// TIA Portal V21 export
FUNCTION "ampoule" : Void   // FC6, LAD
{ S7_Optimized_Access := 'TRUE' }
// stored: SetENOAutomatically false
   VAR_TEMP   // added for the SCL form of the ladder/FBD networks
      _w1 : Bool;
      _w2 : Bool;
   END_VAR
BEGIN

REGION Network 1
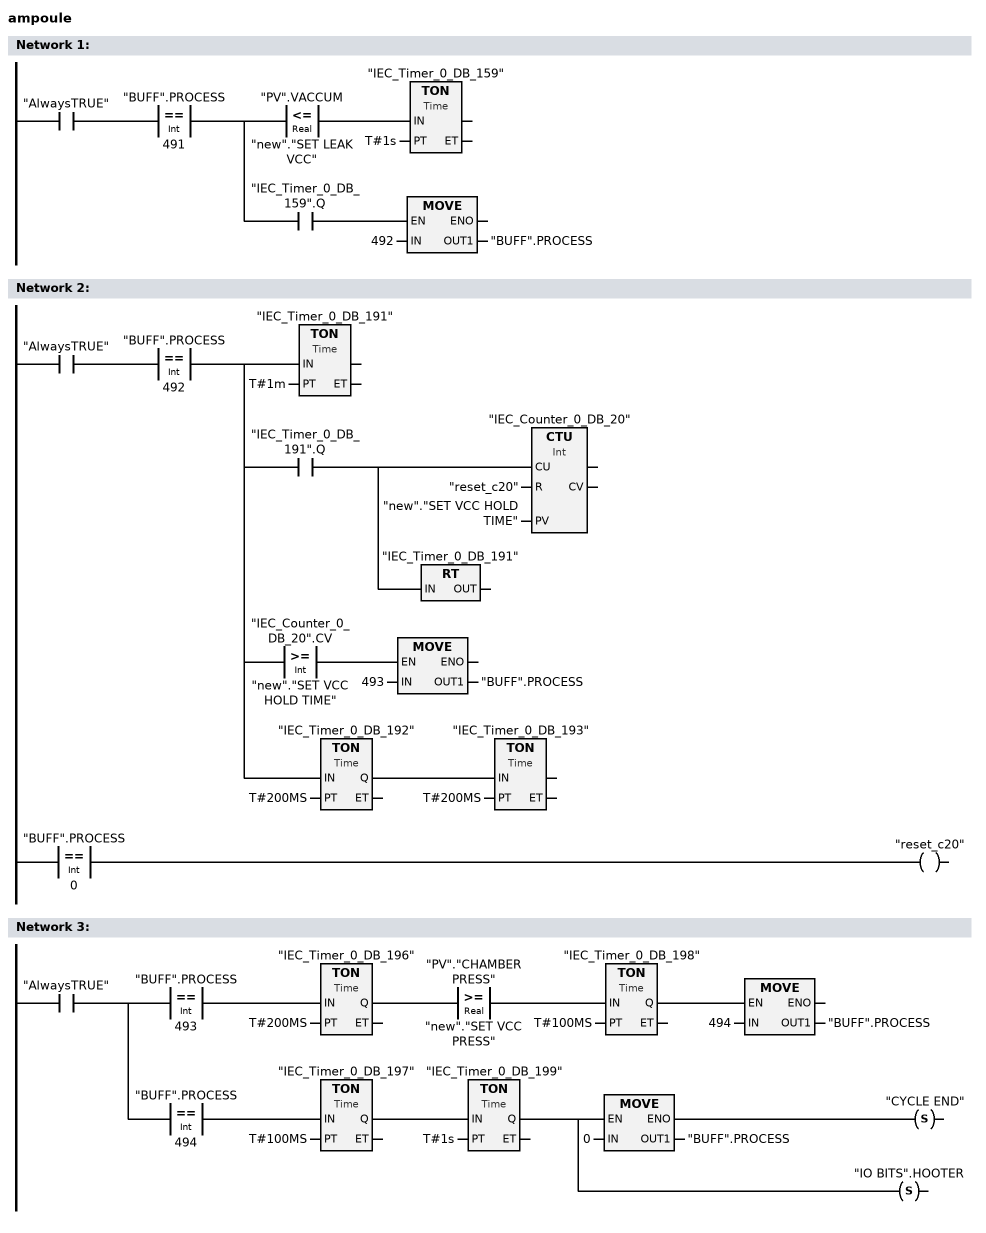
   RUNG wire#powerrail
      Contact( "AlwaysTRUE" )
      { S7_Templates := "SrcType := Int" } EQ_Contact(in1 := "BUFF".PROCESS, in2 := 491)
      wire#w1
      { S7_Templates := "SrcType := Real" } LE_Contact(in1 := "PV".VACCUM, in2 := "new"."SET LEAK VCC")
      { S7_Templates := "time_type := Time" } "IEC_Timer_0_DB_159".TON(pt := T#1s, et =>)
   END_RUNG
   RUNG wire#w1
      Contact( "IEC_Timer_0_DB_159".Q )
      Move(in := 492, out1 => "BUFF".PROCESS)
   END_RUNG
   // the same network as SCL:
   #_w1 := "AlwaysTRUE" AND ("BUFF".PROCESS = 491);
   "IEC_Timer_0_DB_159".TON(IN := #_w1 AND ("PV".VACCUM <= "new"."SET LEAK VCC"), PT := T#1s);
   IF #_w1 AND "IEC_Timer_0_DB_159".Q THEN "BUFF".PROCESS := 492; END_IF;
END_REGION

REGION Network 2
   RUNG wire#powerrail
      Contact( "AlwaysTRUE" )
      { S7_Templates := "SrcType := Int" } EQ_Contact(in1 := "BUFF".PROCESS, in2 := 492)
      wire#w1
      { S7_Templates := "time_type := Time" } "IEC_Timer_0_DB_191".TON(pt := T#1m, et =>)
   END_RUNG
   RUNG wire#w1
      Contact( "IEC_Timer_0_DB_191".Q )
      wire#w2
      { S7_Templates := "value_type := Int" } "IEC_Counter_0_DB_20".CTU(r := "reset_c20", pv := "new"."SET VCC HOLD TIME", cv =>)
   END_RUNG
   RUNG wire#w2
      RT_Coil( "IEC_Timer_0_DB_191" )
   END_RUNG
   RUNG wire#w1
      { S7_Templates := "SrcType := Int" } GE_Contact(in1 := "IEC_Counter_0_DB_20".CV, in2 := "new"."SET VCC HOLD TIME")
      Move(in := 493, out1 => "BUFF".PROCESS)
   END_RUNG
   RUNG wire#w1
      { S7_Templates := "time_type := Time" } "IEC_Timer_0_DB_192".TON(pt := T#200MS, et =>)
      { S7_Templates := "time_type := Time" } "IEC_Timer_0_DB_193".TON(pt := T#200MS, et =>)
   END_RUNG
   RUNG wire#powerrail
      { S7_Templates := "SrcType := Int" } EQ_Contact(in1 := "BUFF".PROCESS, in2 := 0)
      Coil( "reset_c20" )
   END_RUNG
   // the same network as SCL:
   #_w1 := "AlwaysTRUE" AND ("BUFF".PROCESS = 492);
   "IEC_Timer_0_DB_191".TON(IN := #_w1, PT := T#1m);
   #_w2 := #_w1 AND "IEC_Timer_0_DB_191".Q;
   "IEC_Counter_0_DB_20".CTU(CU := #_w2, R := "reset_c20", PV := "new"."SET VCC HOLD TIME");
   IF #_w2 THEN RESET_TIMER("IEC_Timer_0_DB_191"); END_IF;
   IF #_w1 AND ("IEC_Counter_0_DB_20".CV >= "new"."SET VCC HOLD TIME") THEN "BUFF".PROCESS := 493; END_IF;
   "IEC_Timer_0_DB_192".TON(IN := #_w1, PT := T#200MS);
   "IEC_Timer_0_DB_193".TON(IN := "IEC_Timer_0_DB_192".Q, PT := T#200MS);
   "reset_c20" := "BUFF".PROCESS = 0;
END_REGION

REGION Network 3
   RUNG wire#powerrail
      Contact( "AlwaysTRUE" )
      wire#w1
      { S7_Templates := "SrcType := Int" } EQ_Contact(in1 := "BUFF".PROCESS, in2 := 493)
      { S7_Templates := "time_type := Time" } "IEC_Timer_0_DB_196".TON(pt := T#200MS, et =>)
      { S7_Templates := "SrcType := Real" } GE_Contact(in1 := "PV"."CHAMBER PRESS", in2 := "new"."SET VCC PRESS")
      { S7_Templates := "time_type := Time" } "IEC_Timer_0_DB_198".TON(pt := T#100MS, et =>)
      Move(in := 494, out1 => "BUFF".PROCESS)
   END_RUNG
   RUNG wire#w1
      { S7_Templates := "SrcType := Int" } EQ_Contact(in1 := "BUFF".PROCESS, in2 := 494)
      { S7_Templates := "time_type := Time" } "IEC_Timer_0_DB_197".TON(pt := T#100MS, et =>)
      { S7_Templates := "time_type := Time" } "IEC_Timer_0_DB_199".TON(pt := T#1s, et =>)
      wire#w2
      Move(in := 0, out1 => "BUFF".PROCESS)
      S_Coil( "CYCLE END" )
   END_RUNG
   RUNG wire#w2
      S_Coil( "IO BITS".HOOTER )
   END_RUNG
   // the same network as SCL:
   "IEC_Timer_0_DB_196".TON(IN := "AlwaysTRUE" AND ("BUFF".PROCESS = 493), PT := T#200MS);
   "IEC_Timer_0_DB_198".TON(IN := "IEC_Timer_0_DB_196".Q AND ("PV"."CHAMBER PRESS" >= "new"."SET VCC PRESS"),
                           PT := T#100MS);
   IF "IEC_Timer_0_DB_198".Q THEN "BUFF".PROCESS := 494; END_IF;
   "IEC_Timer_0_DB_197".TON(IN := "AlwaysTRUE" AND ("BUFF".PROCESS = 494), PT := T#100MS);
   "IEC_Timer_0_DB_199".TON(IN := "IEC_Timer_0_DB_197".Q, PT := T#1s);
   IF "IEC_Timer_0_DB_199".Q THEN
       "BUFF".PROCESS := 0;
       "CYCLE END" := TRUE;
       "IO BITS".HOOTER := TRUE;
   END_IF;
END_REGION
END_FUNCTION
